PROGRAM MAIN
VAR
END_VAR

END_PROGRAM

(* stored: Version 1.1.0.1
   POU MAIN: Id {72ca4819-2207-4b0a-96f2-921b12ac7780} *)
